// TIA Portal V20 export
// export: Created 2025-12-01T14:57:14.997586Z, ExportSetting None, DisplayName Totally Integrated Automation Portal, DisplayVersion V20 Update 3, DisplayName TIA Portal Openness, DisplayVersion V20 Update 3, DisplayName TIA Portal Version Control Interface, DisplayVersion V20 Update 3, DisplayName STEP 7 Professional, DisplayVersion V20 Update 3, DisplayName STEP 7 Safety, DisplayVersion V20 Update 2, DisplayName WinCC Basic/Comfort/Advanced, DisplayVersion V20 Update 3, DisplayName WinCC Professional, DisplayVersion V20 Update 3, DisplayName WinCC Unified, DisplayVersion V20 Update 3
FUNCTION_BLOCK "FB989_Envio Datos Movimot Asi"   // FB989, SCL
{ S7_Optimized_Access := 'FALSE' }
VERSION : 0.0
// Parámetros del bloque
// stored: AutoNumber false, SetENOAutomatically false
   VAR_INPUT
      Dir_GW_ASI_Com : Int;   // Direccion de inicio de Command Interface del Gateway ASI de Bihl+Wiedemann
      Num_Line : Int;
      Num_Slave : Int;
      Valor_V1 : Real;   // Porcentaje de velocidad respecto de la maxima en formato REAL
      Valor_V2 : Real;
      Valor_V3 : Real;
      Valor_V4 : Real;
      Valor_V5 : Real;
      Valor_V6 : Real;
      Valor_V7 : Real;
      Valor_Rampa : Int;   // Rampa de aceleración en milisegundos
      Escritura : Bool;
      Solo_Velocidades : Bool;
      Solo_Rampa : Bool;
   END_VAR
   VAR_OUTPUT
      Finalizado : Bool;
      Con_Error : Bool;
   END_VAR
   VAR
      Lista_ComVel : Array[1..33] of Byte;
      Lista_ComRampa : Array[1..8] of Byte;
      Escritura_OLD : Bool;
      Ciclo_envio : Int;
   END_VAR
   VAR_TEMP
      Valor_W : Int;
      Valor_B AT Valor_W : Struct
         high : Byte;
         low : Byte;
      END_STRUCT;
      Flanco_Escritura : Bool;
      i : Int;
   END_VAR
BEGIN


       // Área de instrucciones
       #Flanco_Escritura := #Escritura AND NOT #Escritura_OLD ;


       IF #Flanco_Escritura THEN

           //cabecera envio Velocidades
           #Lista_ComVel[1] := 16#7D ;
           #Lista_ComVel[2] := INT_TO_BYTE (#Num_Line - 1);
           #Lista_ComVel[3] := 16#0A ;
           #Lista_ComVel[4] := INT_TO_BYTE (#Num_Slave);  //Num Esclavo ASI
           #Lista_ComVel[5] := 16#0A ;
           //velocidades (nos deben meter un porcentaje, y nosotros ajustar para que el 100.0% sea 16#4000, que en decimal es 16384, y /100=163.84)
           (* classic code: #Valor_W := REAL_TO_INT (#Valor_V1 * 163.84) ;*)
           #Valor_W := REAL_TO_INT (#Valor_V1 * REAL#163.84) ;
           #Lista_ComVel[6] := #Valor_B.high ;
           #Lista_ComVel[7] := #Valor_B.low ;
           #Valor_W := #Valor_W * (-1);
           #Lista_ComVel[8] := #Valor_B.high ;
           #Lista_ComVel[9] := #Valor_B.low ;
           (* classic code: #Valor_W := REAL_TO_INT (#Valor_V2 * 163.84) ;*)
           #Valor_W := REAL_TO_INT (#Valor_V2 * REAL#163.84) ;
           #Lista_ComVel[10] := #Valor_B.high ;
           #Lista_ComVel[11] := #Valor_B.low ;
           #Valor_W := #Valor_W * (-1);
           #Lista_ComVel[12] := #Valor_B.high ;
           #Lista_ComVel[13] := #Valor_B.low ;
           (* classic code: #Valor_W := REAL_TO_INT (#Valor_V3 * 163.84) ;*)
           #Valor_W := REAL_TO_INT (#Valor_V3 * REAL#163.84) ;
           #Lista_ComVel[14] := #Valor_B.high ;
           #Lista_ComVel[15] := #Valor_B.low ;
           #Valor_W := #Valor_W * (-1);
           #Lista_ComVel[16] := #Valor_B.high ;
           #Lista_ComVel[17] := #Valor_B.low ;
           (* classic code: #Valor_W := REAL_TO_INT (#Valor_V4 * 163.84) ;*)
           #Valor_W := REAL_TO_INT (#Valor_V4 * REAL#163.84) ;
           #Lista_ComVel[18] := #Valor_B.high ;
           #Lista_ComVel[19] := #Valor_B.low ;
           #Valor_W := #Valor_W * (-1);
           #Lista_ComVel[20] := #Valor_B.high ;
           #Lista_ComVel[21] := #Valor_B.low ;
           (* classic code: #Valor_W := REAL_TO_INT (#Valor_V5 * 163.84) ;*)
           #Valor_W := REAL_TO_INT (#Valor_V5 * REAL#163.84) ;
           #Lista_ComVel[22] := #Valor_B.high ;
           #Lista_ComVel[23] := #Valor_B.low ;
           #Valor_W := #Valor_W * (-1);
           #Lista_ComVel[24] := #Valor_B.high ;
           #Lista_ComVel[25] := #Valor_B.low ;
           (* classic code: #Valor_W := REAL_TO_INT (#Valor_V6 * 163.84) ;*)
           #Valor_W := REAL_TO_INT (#Valor_V6 * REAL#163.84) ;
           #Lista_ComVel[26] := #Valor_B.high ;
           #Lista_ComVel[27] := #Valor_B.low ;
           #Valor_W := #Valor_W * (-1);
           #Lista_ComVel[28] := #Valor_B.high ;
           #Lista_ComVel[29] := #Valor_B.low ;
           (* classic code: #Valor_W := REAL_TO_INT (#Valor_V7 * 163.84) ;*)
           #Valor_W := REAL_TO_INT (#Valor_V7 * REAL#163.84) ;
           #Lista_ComVel[30] := #Valor_B.high ;
           #Lista_ComVel[31] := #Valor_B.low ;
           #Valor_W := #Valor_W * (-1);
           #Lista_ComVel[32] := #Valor_B.high ;
           #Lista_ComVel[33] := #Valor_B.low ;

           //cabecera envio Rampa
           #Lista_ComRampa[1] := 16#7D ;
           #Lista_ComRampa[2] := INT_TO_BYTE (#Num_Line - 1) ;
           #Lista_ComRampa[3] := 16#0B ;
           #Lista_ComRampa[4] := INT_TO_BYTE (#Num_Slave);  //Num Esclavo ASI
           #Lista_ComRampa[5] := 16#0A ;
           #Lista_ComRampa[6] := 16#0E ;
           //Rampa (nos deben meter la rampa en milisegundos (tiempo para ir de 0 a 50Hz), solo miramos que no sea negativa)
           #Valor_W := ABS (#Valor_Rampa) ;
           #Lista_ComRampa[7] := #Valor_B.high ;
           #Lista_ComRampa[8] := #Valor_B.low ;

           IF #Solo_Rampa THEN
               #Ciclo_envio := 4 ;
           ELSE 
               #Ciclo_envio := 1 ;
           END_IF;

           #Con_Error := false ;

       END_IF;

       IF NOT #Escritura THEN
           #Ciclo_envio := 0 ;
       END_IF;

       CASE #Ciclo_envio OF
           1 :
               // ESCRITURA COMANDO DE VELOCIDADES
               (* classic code: %AB (#Dir_GW_ASI_Com):P := #Lista_ComVel[1];*)
               POKE(area:=16#02,dbNumber:=0,byteOffset:=#Dir_GW_ASI_Com,value:=#Lista_ComVel[1])  ;
               FOR #i := 2 TO 32 BY 1 DO    //copiamos todo
                   (* classic code: %AB (#Dir_GW_ASI_Com + #i):P := #Lista_ComVel[#i + 1];*)
                   POKE(area:=16#02,dbNumber:=0,byteOffset:=#Dir_GW_ASI_Com + #i,value:=#Lista_ComVel[#i + 1])  ;
               END_FOR;

               #Ciclo_envio := 2 ;

           2 :
               // ENVIO COMANDO DE VELOCIDADES
               (* classic code: #Lista_ComVel[2] := #Lista_ComVel[2] OR (%EB (#Dir_GW_ASI_Com + 1):P AND 16#80 ) XOR 16#80;*)
               #Lista_ComVel[2] := #Lista_ComVel[2] OR (PEEK_BYTE(area:=16#01,dbNumber:=0,byteOffset:=#Dir_GW_ASI_Com + 1) AND 16#80 ) XOR 16#80;  //Con el AND miro el bit de toogle en entradas, y lo invierto con el XOR, para despues añadirlo con el OR al comando ya calculado 
               (* classic code: %AB (#Dir_GW_ASI_Com + 1):P := #Lista_ComVel[2];*)
               POKE(area:=16#02,dbNumber:=0,byteOffset:=#Dir_GW_ASI_Com + 1,value:=#Lista_ComVel[2])  ;    //Me guardo el comando completo para saber luego que valor hemos enviado en Toogle

               #Ciclo_envio := 3 ;

           3 :
               // COMPROBAR RESPUESTA A COMANDO DE VELOCIDADES
               (* classic code: IF (%EB (#Dir_GW_ASI_Com + 1):P AND 16#80) = (#Lista_ComVel[2] AND 16#80) THEN*)
               IF (PEEK_BYTE(area:=16#01,dbNumber:=0,byteOffset:=#Dir_GW_ASI_Com + 1) AND 16#80) = (#Lista_ComVel[2] AND 16#80) THEN    //Miro si ha cambiado el Toogle
                   (* classic code: IF (%EB (#Dir_GW_ASI_Com):P = #Lista_ComVel[1]) AND (%EB (#Dir_GW_ASI_Com + 2):P = #Lista_ComVel[3]) THEN*)
                   IF (PEEK_BYTE(area:=16#01,dbNumber:=0,byteOffset:=#Dir_GW_ASI_Com) = #Lista_ComVel[1]) AND (PEEK_BYTE(area:=16#01,dbNumber:=0,byteOffset:=#Dir_GW_ASI_Com + 2) = #Lista_ComVel[3]) THEN   //Miro si el comando de vuelta es igual
                       IF #Solo_Velocidades THEN
                           #Ciclo_envio := 0 ;  //se ha ejecutado el envio correctamente y no hay que enviar rampa
                       ELSE
                           #Ciclo_envio := 4 ;  //se ha ejecutado el envio correctamente y pasamos a enviar rampa 
                       END_IF; 
                       #Con_Error := false ;
                   ELSE
                       #Ciclo_envio := 0 ;  //NO se ha ejecutado el envio correctamente
                       #Con_Error := true ;
                   END_IF;
               END_IF;

           4 :
               // ESCRITURA COMANDO DE RAMPA

               (* classic code: %AB (#Dir_GW_ASI_Com):P := #Lista_ComRampa[1];*)
               POKE(area:=16#02,dbNumber:=0,byteOffset:=#Dir_GW_ASI_Com,value:=#Lista_ComRampa[1])  ;
               FOR #i := 2 TO 7 BY 1 DO    //copiamos todo
                   (* classic code: %AB (#Dir_GW_ASI_Com + #i):P := #Lista_ComRampa[#i + 1];*)
                   POKE(area:=16#02,dbNumber:=0,byteOffset:=#Dir_GW_ASI_Com + #i,value:=#Lista_ComRampa[#i + 1])  ;
               END_FOR;

               #Ciclo_envio := 5 ;

           5 :
               // ENVIO COMANDO DE RAMPA
               (* classic code: #Lista_ComRampa[2] := #Lista_ComRampa[2] OR (%EB (#Dir_GW_ASI_Com + 1):P AND 16#80 ) XOR 16#80;*)
               #Lista_ComRampa[2] := #Lista_ComRampa[2] OR (PEEK_BYTE(area:=16#01,dbNumber:=0,byteOffset:=#Dir_GW_ASI_Com + 1) AND 16#80 ) XOR 16#80;  //Con el AND miro el bit de toogle en entradas, y lo invierto con el XOR, para despues añadirlo con el OR al comando ya calculado 
               (* classic code: %AB (#Dir_GW_ASI_Com + 1):P := #Lista_ComRampa[2];*)
               POKE(area:=16#02,dbNumber:=0,byteOffset:=#Dir_GW_ASI_Com + 1,value:=#Lista_ComRampa[2])  ;    //Me guardo el comando completo para saber luego que valor hemos enviado en Toogle

               #Ciclo_envio := 6 ;

           6 :
               // COMPROBAR RESPUESTA A COMANDO DE RAMPA
               (* classic code: IF (%EB (#Dir_GW_ASI_Com + 1):P AND 16#80) = (#Lista_ComRampa[2] AND 16#80) THEN*)
               IF (PEEK_BYTE(area:=16#01,dbNumber:=0,byteOffset:=#Dir_GW_ASI_Com + 1) AND 16#80) = (#Lista_ComRampa[2] AND 16#80) THEN    //Miro si ha cambiado el Toogle
                   (* classic code: IF (%EB (#Dir_GW_ASI_Com):P = #Lista_ComRampa[1]) AND (%EB (#Dir_GW_ASI_Com + 2):P = #Lista_ComRampa[3]) THEN*)
                   IF (PEEK_BYTE(area:=16#01,dbNumber:=0,byteOffset:=#Dir_GW_ASI_Com) = #Lista_ComRampa[1]) AND (PEEK_BYTE(area:=16#01,dbNumber:=0,byteOffset:=#Dir_GW_ASI_Com + 2) = #Lista_ComRampa[3]) THEN   //Miro si el comando de vuelta es igual
                       #Con_Error := false ;
                   ELSE 
                       #Con_Error := true ;  //NO se ha ejecutado el envio correctamente
                   END_IF;
               #Ciclo_envio := 0 ;
               END_IF;

       ELSE:
           // REPOSO, normalmente Ciclo_envio = 0, pero para cualquier otro caso no contemplado hacemos lo mismo
           #Ciclo_envio := 0 ;
           #Finalizado := #Escritura;
       END_CASE;

       IF NOT #Escritura THEN 
                   (* classic code: %AB (#Dir_GW_ASI_Com):P := 16#00 ;*)
                   POKE(area:=16#02,dbNumber:=0,byteOffset:=#Dir_GW_ASI_Com,value:=DINT_TO_BYTE(16#00))   ;
                   (* classic code: %AB (#Dir_GW_ASI_Com + 2):P := 16#00 ;*)
                   POKE(area:=16#02,dbNumber:=0,byteOffset:=#Dir_GW_ASI_Com + 2,value:=DINT_TO_BYTE(16#00))   ;
                   (* classic code: %AB (#Dir_GW_ASI_Com + 1):P := %EB (#Dir_GW_ASI_Com + 1):P ;*)
                   POKE(area:=16#02,dbNumber:=0,byteOffset:=#Dir_GW_ASI_Com + 1,value:=PEEK_BYTE(area:=16#01,dbNumber:=0,byteOffset:=#Dir_GW_ASI_Com + 1))   ;
       END_IF ;

    //   FOR i := 1 TO 255 BY 1 DO    //para rellenar el DB1000 todo como el Movimot[0]
    //       "Conf_Movimot".Movimot[i]:="Conf_Movimot".Movimot[0];
    //   END_FOR;

       #Escritura_OLD := #Escritura;
END_FUNCTION_BLOCK
